PROGRAM MAIN
VAR
	
bAlwaysTrue  	AT%Q* 	: BOOL := TRUE;
bRun 		 	AT%Q* 	: BOOL;
bErrAck 		AT%Q*	: BOOL;

END_VAR

END_PROGRAM

(* stored: Version 1.1.0.1, ProductVersion 3.1.4024.13
   POU MAIN: Id {2de65154-975d-4f1a-b566-e7882660a616}, SpecialFunc None *)
